Fanuc KAREL source: kb00067.KL

-- PROVISIONAL review KL for V770-1; original PC SHA256 d475d53452bd56d0174a12a56e4412bff833e3c4b63354c735d8af2f0f82eded
-- Incomplete behavior may be omitted. Consult companion uncertainty JSON. Do not deploy.
PROGRAM KB00067
%NOLOCKGROUP
BEGIN
  -- UNRESOLVED_PC offsets 5-14; opcodes 3F,75
  -- UNRESOLVED_PC offsets 19-26; opcodes 9D,23
  -- UNRESOLVED_PC offsets 31-38; opcodes 9D,23
  -- UNRESOLVED_PC offsets 43-50; opcodes 9D,23
  -- UNRESOLVED_PC offsets 55-62; opcodes 9D,23
  -- UNRESOLVED_PC offsets 67-103; opcodes 27,22,2A,22,22,22,22,31
  -- UNRESOLVED_PC offsets 108-112; opcodes 7F
END KB00067
